Fanuc KAREL source: compact_preamble.KL

PROGRAM NC0057
%NOLOCKGROUP
ROUTINE R
VAR
S1:INTEGER
BEGIN
S1=1
SELECT S1 OF
CASE(1):
S1=(S1 + 2)
CASE(2):
S1=(S1 + 3)
ELSE:
IF (S1=1) THEN
S1=(S1 + 2)
ELSE
SELECT S1 OF
CASE(1):
S1=(S1 + 2)
CASE(2):
S1=(S1 + 3)
ELSE:
IF (S1=1) THEN
S1=(S1 + 2)
ELSE
SELECT S1 OF
CASE(1):
S1=(S1 + 2)
CASE(2):
S1=(S1 + 3)
ELSE:
IF (S1=1) THEN
S1=(S1 + 2)
ELSE
SELECT S1 OF
CASE(1):
S1=(S1 + 2)
CASE(2):
S1=(S1 + 3)
ELSE:
IF (S1=1) THEN
S1=(S1 + 2)
ELSE
SELECT S1 OF
CASE(1):
S1=(S1 + 2)
CASE(2):
S1=(S1 + 3)
ELSE:
IF (S1=1) THEN
S1=(S1 + 2)
ELSE
S1=(S1 + 1)
ENDIF
ENDSELECT
ENDIF
ENDSELECT
ENDIF
ENDSELECT
ENDIF
ENDSELECT
ENDIF
ENDSELECT
END R
BEGIN
R
END NC0057
